Yaskawa INFORM job: 947334-U.JBI

/JOB
//NAME 947334-U
//POS
///NPOS 121,0,121,0,0,0
///TOOL 0
///POSTYPE PULSE
///PULSE
C00000=-162679,-31839,-85956,16495,-93507,-72842
C00001=-100204,-31839,-59782,16495,-93507,-24001
C00002=-69279,-31839,-59782,-45071,-78964,49592
C00003=-39089,-9945,-93080,-67851,-46231,57497
C00004=-38754,-6808,-95427,-72704,-45180,60176
C00005=-47804,-29839,-82636,-55348,-58469,51244
C00006=-47804,-45497,-64971,-48412,-70534,43807
C00007=25038,50753,16697,-48014,-58730,37727
C00008=26283,80515,-2619,-57980,-56296,55362
C00009=26729,84018,-5780,-60347,-54110,57063
C00010=26729,47291,8137,-48752,-70787,45699
C00011=-44903,-15291,-39055,-48752,-70787,45699
C00012=-106160,-45717,-71076,-170,-86925,5813
C00013=-162679,-31839,-85956,16495,-93507,-72842
C00014=-162679,-31839,-85956,16495,-93507,-72842
C00015=-80851,-41268,-59179,5939,-69009,-32860
C00016=14265,-52500,-59179,5939,-74567,-69277
C00017=34976,-26297,-75892,8729,-53947,-82905
C00018=36112,-1751,-69033,9870,-45764,-84083
C00019=35706,116,-68424,9965,-45151,-84009
C00020=37380,-21684,-66757,8434,-57381,-83457
C00021=53668,3111,-46866,-623,-57129,-103254
C00022=50798,21214,-48211,-747,-47019,-102206
C00023=50403,22999,-47264,-756,-46687,-102070
C00024=54530,12812,-49561,-669,-50480,-103511
C00025=37356,-29536,-49057,-690,-67289,-18230
C00026=37356,-29536,-49057,-690,-67289,-18230
C00027=22559,6295,-19092,-25200,-77549,52696
C00028=26194,36689,-25464,-38815,-67054,57647
C00029=25497,43984,-27984,-40137,-63160,59479
C00030=24980,42373,-31573,-43343,-60150,61806
C00031=24815,42579,-31127,-42701,-59445,61837
C00032=22683,51960,-19893,-38226,-62181,60378
C00033=22308,52841,-18571,-38017,-62598,60351
C00034=22217,37376,-9045,-34863,-73878,56400
C00035=22173,-28172,-45889,-485,-79152,83688
C00036=27711,9446,-20304,-44497,-63017,41074
C00037=31636,19976,-47180,-56728,-46675,49477
C00038=31910,27581,-45701,-58406,-46912,49923
C00039=27167,23253,-49942,-57341,-48799,50923
C00040=26696,9629,-40665,-49958,-54737,46201
C00041=30205,-22505,-62141,-4114,-69774,77063
C00042=36216,5298,-62285,-5468,-47902,84232
C00043=35592,9244,-60541,-9849,-45730,88971
C00044=40186,8491,-60511,-2965,-46066,74167
C00045=34608,2688,-65585,-4955,-45801,69859
C00046=33979,2167,-65968,-4512,-45990,69933
C00047=29256,15541,-52827,-8928,-60937,72499
C00048=23880,-24068,-59684,-5397,-77808,72684
C00049=36339,-8882,-48365,-4659,-55404,30902
C00050=42899,47288,-1175,-6068,-58492,28179
C00051=42899,56471,-7637,-6757,-49849,28714
C00052=41833,57002,-10984,-5197,-46351,21837
C00053=40960,57042,-12210,-4547,-45263,19464
C00054=40632,58543,-10516,-6281,-46447,25697
C00055=39499,61921,-6540,-1880,-45552,11388
C00056=38524,63929,-4255,3723,-46664,-361
C00057=38073,63825,-5083,9934,-49038,-1752
C00058=40750,64241,-969,12210,-49145,-3260
C00059=42090,47568,9174,9002,-62997,-2025
C00060=35246,-1304,-13979,9002,-62997,-2025
C00061=-16907,-24566,-33119,9002,-62997,-17053
C00062=-12369,1441,-37817,14671,-61073,-53928
C00063=-8695,7384,-50860,-1965,-43806,-45614
C00064=-3697,11213,-51398,1952,-41496,-53971
C00065=-2987,12738,-50807,2101,-41087,-54261
C00066=-5590,7865,-51564,1548,-43078,-53192
C00067=-8441,31371,-29602,-7429,-46237,-32478
C00068=-4972,34037,-29204,-4657,-44395,-28811
C00069=-6765,33780,-25712,-2262,-47891,-28940
C00070=-4199,35044,-27819,-1992,-45891,-29857
C00071=-4186,33671,-29039,-1991,-45840,-29863
C00072=-2978,22802,-39676,2704,-40517,-31482
C00073=-3101,20483,-42090,3335,-40161,-34289
C00074=-5927,20788,-39855,-1025,-43966,-29490
C00075=-19758,-3501,-4648,-2432,-78383,-24991
C00076=-13859,-6430,-7016,-1714,-78278,-27022
C00077=-4234,-5020,-26751,4472,-73359,-37209
C00078=-3464,4192,-39507,4899,-60861,-37967
C00079=-2485,4363,-40655,4946,-60122,-38337
C00080=-2522,1786,-42851,4947,-60093,-38326
C00081=-2569,-175,-44664,5018,-60416,-40993
C00082=-6122,937,-31875,4705,-67494,-39477
C00083=8713,26571,15970,4453,-84535,-43896
C00084=25873,33447,20989,-1007,-73135,-25130
C00085=26659,34266,2138,-965,-61106,-25315
C00086=29967,43100,-5031,4147,-61923,-25645
C00087=30479,45833,-5572,3230,-64773,-26916
C00088=30364,49583,-3093,-547,-65407,-27563
C00089=30691,48542,-4249,66,-65258,-24619
C00090=30224,49606,-2475,405,-65785,-22987
C00091=29852,46342,5865,1796,-70157,-23081
C00092=27903,50935,38704,1761,-87957,-22171
C00093=-4614,19310,17376,2504,-90204,-34306
C00094=-4614,19310,17376,2504,-90204,-34306
C00095=-14071,22518,-30855,1723,-57599,-40334
C00096=-4376,24350,-50388,3799,-48549,-41406
C00097=-3441,23608,-52479,3583,-46587,-43017
C00098=-3411,25949,-50100,3566,-46850,-43016
C00099=-3445,26588,-49558,3568,-46854,-43005
C00100=-7322,28825,-42901,1933,-50836,-39800
C00101=-15505,10215,-10262,1953,-80298,-36621
C00102=14882,10215,11883,1953,-69170,7579
C00103=14881,10215,11882,1953,-69171,7575
C00104=8933,24364,-18071,-23460,-81900,40929
C00105=11334,3303,-52651,-8276,-76197,61974
C00106=9899,2540,-54910,-7875,-74957,62463
C00107=10308,-1897,-58968,-7424,-69103,62495
C00108=7337,-2101,-59951,-6755,-68817,63381
C00109=7266,-621,-57442,-6913,-73035,63255
C00110=14032,3955,-49424,-8649,-75052,61154
C00111=9420,28261,6369,-16542,-91027,47781
C00112=10648,8411,-11782,-12425,-61535,25284
C00113=13297,21266,-31167,7594,-40142,-1367
C00114=12851,30886,-30650,26274,-39623,-9200
C00115=12016,31471,-32214,24116,-40573,-4798
C00116=12396,34493,-29123,19166,-42065,-6579
C00117=12673,31533,-29985,25468,-40715,-14973
C00118=23173,6588,-19493,12720,-58301,-13680
C00119=-31674,-34816,-33158,12720,-58301,-13680
C00120=-162679,-31839,-85956,16495,-93507,-72842
EC00000=-1
EC00001=-1
EC00002=-1
EC00003=-1
EC00004=-1
EC00005=-1
EC00006=-1
EC00007=-1
EC00008=-1
EC00009=-1
EC00010=-1
EC00011=-1
EC00012=-1
EC00013=-1
EC00014=-1
EC00015=-1
EC00016=-1
EC00017=-1
EC00018=-1
EC00019=-1
EC00020=-1
EC00021=-1
EC00022=-1
EC00023=-1
EC00024=-1
EC00025=-1
EC00026=-144392
EC00027=-93701
EC00028=-93699
EC00029=-93699
EC00030=-93699
EC00031=-93699
EC00032=-93699
EC00033=-93699
EC00034=-93699
EC00035=-1185
EC00036=-1185
EC00037=-1186
EC00038=-1186
EC00039=-1186
EC00040=-1186
EC00041=663
EC00042=662
EC00043=662
EC00044=662
EC00045=662
EC00046=662
EC00047=662
EC00048=662
EC00049=-145527
EC00050=-145527
EC00051=-145527
EC00052=-145526
EC00053=-145526
EC00054=-145526
EC00055=-145526
EC00056=-145526
EC00057=-145526
EC00058=-145526
EC00059=-145526
EC00060=-145526
EC00061=-145526
EC00062=-145526
EC00063=-145526
EC00064=-145526
EC00065=-145526
EC00066=-145526
EC00067=-145526
EC00068=-145526
EC00069=-145526
EC00070=-145526
EC00071=-145526
EC00072=-145526
EC00073=-145526
EC00074=-145526
EC00075=-145526
EC00076=-288485
EC00077=-288485
EC00078=-288485
EC00079=-288485
EC00080=-288485
EC00081=-288485
EC00082=-288485
EC00083=-288485
EC00084=-288485
EC00085=-288485
EC00086=-288485
EC00087=-288485
EC00088=-288485
EC00089=-288485
EC00090=-288485
EC00091=-288485
EC00092=-288485
EC00093=-288485
EC00094=952
EC00095=952
EC00096=952
EC00097=952
EC00098=952
EC00099=952
EC00100=952
EC00101=952
EC00102=952
EC00103=146469
EC00104=146469
EC00105=146469
EC00106=146469
EC00107=146469
EC00108=146469
EC00109=146469
EC00110=146469
EC00111=146469
EC00112=-148378
EC00113=-148378
EC00114=-148378
EC00115=-148378
EC00116=-148378
EC00117=-148378
EC00118=-148378
EC00119=-148378
EC00120=-1
//INST
///DATE 2018/02/28 15:08
///ATTR SC,RW
///GROUP1 RB1
///GROUP2 ST1
NOP
JUMP *SPITZE
'SPITZE ROB 1
MOVJ C00000 VJ=100.00  +MOVJ EC00000 VJ=100.00
MOVJ C00001 VJ=100.00  +MOVJ EC00001 VJ=100.00
MOVJ C00002 VJ=100.00  +MOVJ EC00002 VJ=100.00
MOVJ C00003 VJ=100.00  +MOVJ EC00003 VJ=100.00
MOVL C00004 V=8.3 PL=0  +MOVJ EC00004 VJ=100.00
MOVJ C00005 VJ=100.00  +MOVJ EC00005 VJ=100.00
MOVJ C00006 VJ=100.00  +MOVJ EC00006 VJ=100.00
MOVJ C00007 VJ=100.00  +MOVJ EC00007 VJ=100.00
MOVJ C00008 VJ=100.00  +MOVJ EC00008 VJ=100.00
MOVL C00009 V=8.3 PL=0  +MOVJ EC00009 VJ=100.00
MOVJ C00010 VJ=100.00  +MOVJ EC00010 VJ=100.00
MOVJ C00011 VJ=100.00  +MOVJ EC00011 VJ=100.00
MOVJ C00012 VJ=100.00  +MOVJ EC00012 VJ=100.00
MOVJ C00013 VJ=100.00  +MOVJ EC00013 VJ=100.00
*SPITZE
'--------------------------------
'PROGRAMM ERSTELLT(( WEINERT
'DATUM (( 10.02.2018
'--------------------------------
'PROGRAMM  FREIGEGEBEN((
'DATUM((
'--------------------------------
'PROGRAMM  GE�NDERT
'DATUM((
'--------------------------------
'GRUND �NDERUUNG((
'DATUM((
'--------------------------------
'ROB 38
'ROB 1 T-1
'--------------------------------
'321 857 602 041  1.ARBG
'BM NR 933-434
'AE 30
'--------------------------------
MOVJ C00014 VJ=100.00  +MOVJ EC00014 VJ=100.00
MOVJ C00015 VJ=100.00  +MOVJ EC00015 VJ=100.00
TSYNC 1 SNUM=2
MOVJ C00016 VJ=100.00  +MOVJ EC00016 VJ=100.00
DOUT OT#(17) OFF
MOVJ C00017 VJ=100.00  +MOVJ EC00017 VJ=100.00
'2 X HEFTEN
MACRO1 MJ#(0) ARGF2 ARGF4 ARGF0 ARGF0
MOVJ C00018 VJ=100.00  +MOVJ EC00018 VJ=100.00
MOVJ C00019 VJ=100.00  +MOVJ EC00019 VJ=100.00
ARCON
ARCOF
WAIT IN#(35)=OFF
MOVJ C00020 VJ=100.00  +MOVJ EC00020 VJ=100.00
MOVJ C00021 VJ=100.00  +MOVJ EC00021 VJ=100.00
MOVJ C00022 VJ=100.00  +MOVJ EC00022 VJ=100.00
MOVJ C00023 VJ=100.00  +MOVJ EC00023 VJ=100.00
ARCON
ARCOF
WAIT IN#(35)=OFF
WAIT I
MOVJ C00024 VJ=100.00  +MOVJ EC00024 VJ=100.00
MOVJ C00025 VJ=100.00  +MOVJ EC00025 VJ=100.00
TSYNC 2 SNUM=2
MOVJ C00026 VJ=100.00  +MOVJ EC00026 VJ=100.00
TSYNC 3 SNUM=2
TSYNC 4 SNUM=2
MOVJ C00027 VJ=100.00  +MOVJ EC00027 VJ=100.00
TSYNC 5 SNUM=2
MOVJ C00028 VJ=100.00  +MOVJ EC00028 VJ=100.00
'W 19
MACRO1 MJ#(0) ARGF7 ARGF3 ARGF0 ARGF0
MOVJ C00029 VJ=100.00  +MOVJ EC00029 VJ=100.00
MOVJ C00030 VJ=100.00  +MOVJ EC00030 VJ=100.00
ARCON
MOVL C00031 V=12.5  +MOVJ EC00031 VJ=100.00
MOVL C00032 V=10.8  +MOVJ EC00032 VJ=100.00
MOVL C00033 V=10.8  +MOVJ EC00033 VJ=100.00
ARCOF
WAIT IN#(35)=OFF
MOVJ C00034 VJ=100.00  +MOVJ EC00034 VJ=100.00
TSYNC 6 SNUM=2
MOVJ C00035 VJ=100.00  +MOVJ EC00035 VJ=100.00
TSYNC 7 SNUM=2
MOVJ C00036 VJ=100.00  +MOVJ EC00036 VJ=100.00
'W 48
MACRO1 MJ#(0) ARGF7 ARGF3 ARGF0 ARGF0
MOVJ C00037 VJ=100.00  +MOVJ EC00037 VJ=100.00
MOVJ C00038 VJ=100.00  +MOVJ EC00038 VJ=100.00
ARCON
WVON WEV#(5)
MOVL C00039 V=4.0  +MOVJ EC00039 VJ=100.00
ARCOF
WVOF
WAIT IN#(35)=OFF
MOVJ C00040 VJ=100.00  +MOVJ EC00040 VJ=100.00
MOVJ C00041 VJ=100.00  +MOVJ EC00041 VJ=100.00
TSYNC 8 SNUM=2
'W 47
MACRO1 MJ#(0) ARGF7 ARGF3 ARGF0 ARGF0
MOVJ C00042 VJ=100.00  +MOVJ EC00042 VJ=100.00
MOVJ C00043 VJ=100.00  +MOVJ EC00043 VJ=100.00
ARCON
MOVL C00044 V=11.7  +MOVJ EC00044 VJ=100.00
MOVL C00045 V=10.8  +MOVJ EC00045 VJ=100.00
MOVL C00046 V=10.8  +MOVJ EC00046 VJ=100.00
MOVL C00047 V=11.7  +MOVJ EC00047 VJ=100.00
ARCOF

Halllo World

Test

INST

INTERRUPT DECL priority WHEN trigger DO event

WAIT IN#(35)=OFF
MOVJ C00048 VJ=100.00  +MOVJ EC00048 VJ=100.00
TSYNC 9 SNUM=2
MOVJ C00049 VJ=100.00  +MOVJ EC00049 VJ=100.00
MOVJ C00050 VJ=100.00  +MOVJ EC00050 VJ=100.00
MOVJ C00051 VJ=100.00  +MOVJ EC00051 VJ=100.00
'W 20-21
MACRO1 MJ#(0) ARGF7 ARGF3 ARGF0 ARGF0
MOVJ C00052 VJ=100.00  +MOVJ EC00052 VJ=100.00
MOVJ C00053 VJ=100.00  +MOVJ EC00053 VJ=100.00
ARCON
MOVL C00054 V=10.8  +MOVJ EC00054 VJ=100.00
MOVL C00055 V=10.0  +MOVJ EC00055 VJ=100.00
MOVL C00056 V=10.0  +MOVJ EC00056 VJ=100.00
MOVL C00057 V=10.8  +MOVJ EC00057 VJ=100.00
ARCOF
WAIT IN#(35)=OFF
MOVJ C00058 VJ=100.00  +MOVJ EC00058 VJ=100.00
MOVJ C00059 VJ=100.00  +MOVJ EC00059 VJ=100.00
MOVJ C00060 VJ=100.00  +MOVJ EC00060 VJ=100.00
MOVJ C00061 VJ=100.00  +MOVJ EC00061 VJ=100.00
MACRO1 MJ#(4) ARGF2 ARGF1
MACRO1 MJ#(4) ARGF2 ARGF4
MACRO1 MJ#(4) ARGF2 ARGF3
TSYNC 10 SNUM=2
TIMER T=2.00
MOVJ C00062 VJ=100.00  +MOVJ EC00062 VJ=100.00
MOVJ C00063 VJ=100.00  +MOVJ EC00063 VJ=100.00
'W 18
MACRO1 MJ#(0) ARGF2 ARGF5 ARGF0 ARGF0
MOVJ C00064 VJ=100.00  +MOVJ EC00064 VJ=100.00
MOVJ C00065 VJ=100.00  +MOVJ EC00065 VJ=100.00
ARCON
TIMER T=0.30
ARCOF
WAIT IN#(35)=OFF
MOVJ C00066 VJ=100.00  +MOVJ EC00066 VJ=100.00
MOVJ C00067 VJ=100.00  +MOVJ EC00067 VJ=100.00
MOVJ C00068 VJ=100.00  +MOVJ EC00068 VJ=100.00
ARCON
TIMER T=0.50
ARCOF
WAIT IN#(35)=OFF
MOVJ C00069 VJ=100.00  +MOVJ EC00069 VJ=100.00
MACRO1 MJ#(0) ARGF7 ARGF3 ARGF0 ARGF0
MOVJ C00070 VJ=100.00  +MOVJ EC00070 VJ=100.00
ARCON
WVON WEV#(6)
MOVL C00071 V=10.8  +MOVJ EC00071 VJ=100.00
MOVL C00072 V=10.0  +MOVJ EC00072 VJ=100.00
MOVL C00073 V=10.8  +MOVJ EC00073 VJ=100.00
ARCOF
WVOF
WAIT IN#(35)=OFF
MOVJ C00074 VJ=100.00  +MOVJ EC00074 VJ=100.00
MOVJ C00075 VJ=100.00  +MOVJ EC00075 VJ=100.00
TSYNC 11 SNUM=2
MOVJ C00076 VJ=100.00  +MOVJ EC00076 VJ=100.00
TSYNC 12 SNUM=2
MOVJ C00077 VJ=100.00  +MOVJ EC00077 VJ=100.00
'W 9
MOVJ C00078 VJ=100.00  +MOVJ EC00078 VJ=100.00
MOVJ C00079 VJ=100.00  +MOVJ EC00079 VJ=100.00
ARCON
MOVL C00080 V=11.7  +MOVJ EC00080 VJ=100.00
MOVL C00081 V=10.8  +MOVJ EC00081 VJ=100.00
ARCOF
WAIT IN#(35)=OFF
MOVJ C00082 VJ=100.00  +MOVJ EC00082 VJ=100.00
MOVJ C00083 VJ=100.00  +MOVJ EC00083 VJ=100.00
MOVJ C00084 VJ=100.00  +MOVJ EC00084 VJ=100.00
MOVJ C00085 VJ=100.00  +MOVJ EC00085 VJ=100.00
MOVJ C00086 VJ=100.00  +MOVJ EC00086 VJ=100.00
MOVJ C00087 VJ=100.00  +MOVJ EC00087 VJ=100.00
'W 5
MOVJ C00088 VJ=100.00  +MOVJ EC00088 VJ=100.00
ARCON
MOVL C00089 V=11.7  +MOVJ EC00089 VJ=100.00
ARCOF
WAIT IN#(35)=OFF
MOVJ C00090 VJ=100.00  +MOVJ EC00090 VJ=100.00
MOVJ C00091 VJ=100.00  +MOVJ EC00091 VJ=100.00
MOVJ C00092 VJ=100.00  +MOVJ EC00092 VJ=100.00
MOVJ C00093 VJ=100.00  +MOVJ EC00093 VJ=100.00
TSYNC 13 SNUM=2
MOVJ C00094 VJ=100.00  +MOVJ EC00094 VJ=100.00
MACRO1 MJ#(4) ARGF1 ARGF5
TSYNC 25 SNUM=2
MOVJ C00095 VJ=100.00  +MOVJ EC00095 VJ=100.00
'W 8
MOVJ C00096 VJ=100.00  +MOVJ EC00096 VJ=100.00
MOVJ C00097 VJ=100.00  +MOVJ EC00097 VJ=100.00
ARCON
MOVL C00098 V=11.7  +MOVJ EC00098 VJ=100.00
MOVL C00099 V=10.8  +MOVJ EC00099 VJ=100.00
ARCOF
WAIT IN#(35)=OFF
MOVJ C00100 VJ=100.00  +MOVJ EC00100 VJ=100.00
MOVJ C00101 VJ=100.00  +MOVJ EC00101 VJ=100.00
MOVJ C00102 VJ=100.00  +MOVJ EC00102 VJ=100.00
TSYNC 14 SNUM=2
MOVJ C00103 VJ=100.00  +MOVJ EC00103 VJ=100.00
TSYNC 15 SNUM=2
MOVJ C00104 VJ=100.00  +MOVJ EC00104 VJ=100.00
'W 51
MACRO1 MJ#(0) ARGF7 ARGF3 ARGF0 ARGF0
MOVJ C00105 VJ=100.00  +MOVJ EC00105 VJ=100.00
MOVJ C00106 VJ=100.00  +MOVJ EC00106 VJ=100.00
MOVJ C00107 VJ=100.00  +MOVJ EC00107 VJ=100.00
ARCON
TIMER T=0.30
MOVL C00108 V=11.7  +MOVJ EC00108 VJ=100.00
ARCOF
WAIT IN#(35)=OFF
MOVJ C00109 VJ=100.00  +MOVJ EC00109 VJ=100.00
MOVJ C00110 VJ=100.00  +MOVJ EC00110 VJ=100.00
MOVJ C00111 VJ=100.00  +MOVJ EC00111 VJ=100.00
TSYNC 16 SNUM=2
MOVJ C00112 VJ=100.00  +MOVJ EC00112 VJ=100.00
TSYNC 17 SNUM=2
MOVJ C00113 VJ=100.00  +MOVJ EC00113 VJ=100.00
'W 53
DOUT OT#(62) ON
MOVJ C00114 VJ=100.00  +MOVJ EC00114 VJ=100.00
MOVJ C00115 VJ=100.00  +MOVJ EC00115 VJ=100.00
ARCON
TIMER T=0.30
MOVL C00116 V=10.0  +MOVJ EC00116 VJ=100.00
ARCOF
WAIT IN#(35)=OFF
MOVJ C00117 VJ=100.00  +MOVJ EC00117 VJ=100.00
DOUT OT#(62) OFF
MOVJ C00118 VJ=100.00  +MOVJ EC00118 VJ=100.00
MOVJ C00119 VJ=100.00  +MOVJ EC00119 VJ=100.00
TSYNC 18 SNUM=2
MACRO1 MJ#(4) ARGF2 ARGF2
MACRO1 MJ#(4) ARGF0 ARGF2
MACRO1 MJ#(4) ARGF2 ARGF5
MACRO1 MJ#(4) ARGF0 ARGF5
MOVJ C00120 VJ=100.00  +MOVJ EC00120 VJ=100.00
END
